TYPE ST_Configuration :
STRUCT
  XtsStationParameter  : ARRAY[1..MAX_STATION] OF ST_STATION_PARAMETER;
END_STRUCT
END_TYPE

(* stored: Version 1.1.0.1, ProductVersion 3.1.4026.20
   DUT ST_Configuration: Id {a3108960-908c-4395-a04d-33836fdd3ae9} *)
